Staubli VAL3: AtHomePulse.pgx

public program AtHomePulse()
begin

  //2014.12.09
  //回零脉冲
  waitEndMove()
  dDio["UsO_bNull2"]=true
  call Digtal2Analog()
  delay(0.5)
  dDio["UsO_bNull2"]=false
  call Digtal2Analog()


  //信号确认
  delay(0.5)
  dDio["UsO_bNull1"]=true
  delay(0.5)
  dDio["UsO_bNull1"]=false
  delay(0.5)
  dDio["UsO_bNull7"]=true
  delay(0.5)
  dDio["UsO_bNull7"]=false
  delay(0.5)


end
